TYPE
    TcoSmartFunctionKitConfig_v_4_x_x :
    STRUCT
        DataFormat : eTcoDataFormat := TcoUtilities.eTcoDataFormat.BigEndian;
        InfoTime : TIME := T#2S;
        ErrorTime : TIME := T#5S;
		IpAddress : STRING;
		CurveExportLocation : STRING;
    END_STRUCT
END_TYPE

(* stored: Version 1.1.0.1, ProductVersion 3.1.4024.11
   DUT TcoSmartFunctionKitConfig_v_4_x_x: Id {e14a5d54-2aa1-4e00-8fb0-64bc9475e2ad} *)
